(* IEC 61131-3 sources: log21/plc-runtime/plc/edit_plc/prog, 1 file *)

(* ---- bobbio.plc ---- *)
VAR_GLOBAL
	_CREATED : UDINT:= 975945928;
	_VERSION : STRING:= '1.0.0.0';
END_VAR

PROGRAM NONAME

	LD	IN1
	ST	OUT1
	LD	IN2
	ST	OUT2

END_PROGRAM
